DEVICE_TYPE BeagleBoneBlack (* BeagleBoneBlack controller *)
  (* Standard: 61499 ITA; Description: Copyright (c) 2015 fortiss GmbH This program and the accompanying materials are made available under the terms of the Eclipse Public License 2.0 which is available at https://www.eclipse.org/legal/epl-2.0/ SPDX-License-Identifier: EPL-2.0 *)
  (* Version 1.0, 2015-10-31, Alois Zoitl, fortiss GmbH, Initial version *)
  VAR_INPUT
    MGR_ID : WSTRING := "localhost:61499"; (* Device manager socket ID *)
  END_VAR
END_DEVICE_TYPE
